SUBAPPLICATION ROUND_STEP_AR (* Rundet AR_IN auf ein beliebiges Raster RASTER (z.B. 0.25), nicht nur auf Nachkommastellen wie ROUND_AR. Rechenweg: ROUND(AR_IN / RASTER) * RASTER. Vorerst als SUB (wiederverwendet das bestehende ROUND_AR), spaeter ggf. als eigener Basic-Block. *)
  (* Standard: 61499-2; Description: Copyright (c) 2026 Meisterschulen am Ostbahnhof This program and the accompanying materials are made available under the terms of the Eclipse Public License 2.0 which is available at https://www.eclipse.org/legal/epl-2.0/ SPDX-License-Identifier: EPL-2.0 *)
  (* Version 1.1, 2026-10-03, Franz Höpfinger, Meisterschulen am Ostbahnhof, Bugfix (4diac-IDE-Validation: 'Name: STEP is a reserved keyword' - IEC 61131-3 SFC reserviert STEP fuer Schritte in Ablaufsprache): InputVar STEP in RASTER umbenannt. *)
  (* Version 1.0, 2026-10-03, Franz Höpfinger, Meisterschulen am Ostbahnhof, initial implementation - Franz: 'haben wir einen Baustein um z.B. auf 0.25 zu RUNDEN?' - ROUND_AR/RND_AR/CEIL_AR/FLOOR_AR runden nur auf Nachkommastellen bzw. auf ganze Zahlen, keiner davon auf ein beliebiges Raster. Vorerst als SUB (reine Verdrahtung bestehender Bausteine: AR_DIV_2 -> ROUND_AR(N=0) -> AR_MUL_2), spaeter ggf. als eigener Basic-Block. *)
  PACKAGE OSCAT_adapter::Mathematical;
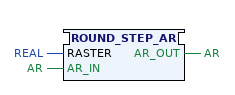
  VAR_INPUT
    RASTER : REAL := 1.0; (* Rundungsraster, z.B. 0.25 - Platzhalter-Default 1.0 (= Rundung auf ganze Zahl), per Parameter ueberschreibbar *)
  END_VAR
  SOCKETS
    AR_IN : adapter::types::unidirectional::AR; (* Eingangssignal (REAL) *)
  END_SOCKETS
  PLUGS
    AR_OUT : adapter::types::unidirectional::AR; (* Auf RASTER gerundeter Wert (REAL) *)
  END_PLUGS
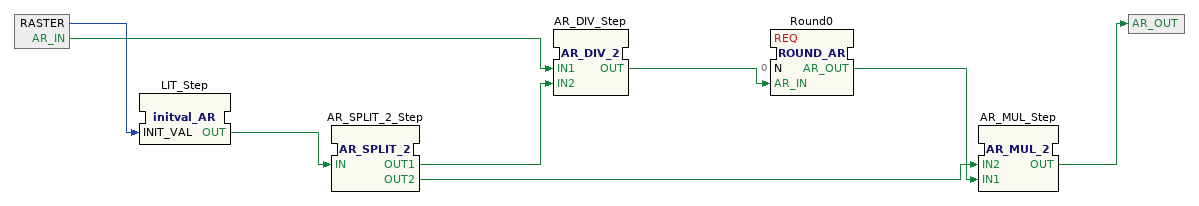
  FBS
    LIT_Step : adapter::types::unidirectional::AR::initval::initval_AR;
    AR_SPLIT_2_Step : adapter::events::unidirectional::AR_SPLIT_2; (* Faechert RASTER auf AR_DIV_Step und AR_MUL_Step auf - Adapter-Fanout ist strikt 1:1. *)
    AR_DIV_Step : adapter::iec61131::arithmetic::AR_DIV_2;
    Round0 : OSCAT_adapter::Mathematical::ROUND_AR(N := 0); (* N=0: rundet den Quotienten auf eine ganze Zahl. *)
    AR_MUL_Step : adapter::iec61131::arithmetic::AR_MUL_2;
  END_FBS
  DATA_CONNECTIONS
    RASTER TO LIT_Step.INIT_VAL;
  END_CONNECTIONS
  ADAPTER_CONNECTIONS
    AR_IN TO AR_DIV_Step.IN1;
    LIT_Step.OUT TO AR_SPLIT_2_Step.IN;
    AR_SPLIT_2_Step.OUT1 TO AR_DIV_Step.IN2;
    AR_SPLIT_2_Step.OUT2 TO AR_MUL_Step.IN2;
    AR_DIV_Step.OUT TO Round0.AR_IN;
    Round0.AR_OUT TO AR_MUL_Step.IN1;
    AR_MUL_Step.OUT TO AR_OUT;
  END_CONNECTIONS
END_SUBAPPLICATION
